FUNCTION_BLOCK FT_PT1 (* Low Pass Filter (PT1) *)
  (* Standard: 61499-1; Description: FT_PT1 is an low pass filter with a programmable time T and faktor K. *)
  (* Version 1.3, 2026-09-26, Franz Höpfinger, Bugfix (Review-Bot auf training1 PR #269, verifiziert): die neue TM.E1->RST-Verdrahtung (FT_PT1_AR v1.0) feuert RST bereits beim Start-Kaskaden-INIT (z.B. ueber initval_ATM/LatchFilterTime.INIT -> OUT.E1 -> TM.E1, siehe logiBUS_PI_Raw_Publish_OPC.SUB), also BEVOR je ein echtes REQ mit frisch abgetastetem 'in' lief. RST setzte bisher init:=TRUE UND out:=K*in mit dem zu diesem Zeitpunkt noch nie gesetzten 'in' (0.0) - das erste echte REQ sah dann init bereits TRUE und ramp'te per Euler-Schritt langsam von 0 auf den echten Wert hoch, statt sofort zu springen. RST setzt jetzt NUR NOCH init:=FALSE (kein 'in'-With-Var, kann also gar nicht sinnvoll seeden) - das naechste REQ (mit garantiert frischem 'in') macht das Seeding selbst inline (vorher this.RST(), jetzt direkt out:=K*in), genau wie beim allerersten Programmstart. *)
  (* Version 1.2, 2026-09-25, Franz Höpfinger, Bugfix (Franz live am Geraet: 'ich hatte von 2s auf 0.1s geaendert, und schwupps spinnt er' - Zapfwelle-Filterzeit auf STG4 manuell auf 100ms gesenkt): die explizite Euler-Diskretisierung wird numerisch instabil, sobald TM kleiner als das tatsaechliche REQ-Aufrufintervall (delta_t) ist - Faktor delta_t/TM > 1 laesst den Fehler pro Zyklus exponentiell wachsen statt sich dem Zielwert anzunaehern, bis out ueberlaeuft (Inf) und danach dauerhaft NaN bleibt (Inf-Inf), da kein automatisches Re-Init/RST mehr verdrahtet war. TM wird in der REQ-Berechnung jetzt adaptiv auf mindestens delta_t hochgeklemmt (Franz' Vorschlag, F1/F2-Notation) - Faktor bleibt so immer <= 1, unabhaengig von der tatsaechlichen Aufrufrate, kein fixer Magic-Number-Mindestwert noetig. *)
  (* Version 1.1, 2026-09-17, Franz Höpfinger, Bugfix (Review-Bot auf training1 PR #252, verifiziert): RST setzte init/out zurueck, aber nicht tx/last/delta_t - ein externer RST-Aufruf (jetzt ueber FT_PT1_AR.RST erreichbar) liess die naechste REQ-Ausfuehrung mit einem stehengebliebenen last einen riesigen delta_t berechnen und dadurch einen falschen Ausreisser-Schritt. RST liest jetzt T_PLC_US() neu und setzt last/delta_t entsprechend zurueck. *)
  (* Version 1.0, 2025-12-21, Franz Höpfinger, initial API and implementation and/or initial documentation *)
  PACKAGE OSCAT::Basic::POUs::Engineering::Control;
  IMPORT OSCAT::Basic::POUs::Engineering::measurements::T_PLC_US;
  IMPORT OSCAT::Basic::POUs::conversion::TIME_TO_REAL;
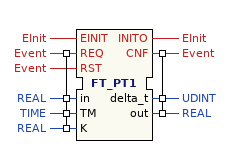
  EVENT_INPUT
    EINIT : EInit; (* Init Request *)
    REQ WITH in, TM, K; (* Normal Execution Request *)
    RST; (* Reset Filter *)
  END_EVENT
  EVENT_OUTPUT
    INITO : EInit; (* Init Confirmation *)
    CNF WITH delta_t, out; (* Execution Confirmation *)
  END_EVENT
  VAR_INPUT
    in : REAL; (* Input Signal *)
    TM : TIME; (* Filter Time Constant *)
    K : REAL := 1.0; (* Gain Factor *)
  END_VAR
  VAR_OUTPUT
    delta_t : UDINT; (* Delta T since last call. *)
    out : REAL; (* Output Signal *)
  END_VAR
  VAR
    last : UDINT; (* Last execution time *)
    tx : UDINT; (* Current execution time *)
    init : BOOL := FALSE; (* Initialization flag *)
    F1 : REAL;
    F2 : REAL;
  END_VAR
  EC_STATES
    EINIT : EINIT -> INITO; (* Initialization *)
    REQ : REQ -> CNF; (* Normal Operation *)
    RST : RST -> CNF;
  END_STATES
  ALGORITHM EINIT IN ST:
(* Reset logic *)
init := FALSE;
out := 0.0;
last := UDINT#0;
  END_ALGORITHM
  ALGORITHM RST IN ST:
(* Nur den Zustand invalidieren - das naechste REQ seedet mit frisch
   abgetastetem 'in' (With-Var, synchron zum REQ-Event). RST selbst hat
   kein 'in'-With-Var und wuerde sonst mit einem veralteten oder (beim
   allerersten Aufruf, z.B. durch TM.E1 vor der ersten echten Messung)
   noch nie gesetzten Wert (0.0) faelschlich seeden. *)
init := FALSE;
  END_ALGORITHM
  ALGORITHM REQ IN ST:
(* Read system time *)
tx := T_PLC_US();

(* Startup initialization or T=0 *)
IF NOT init OR TM = T#0s THEN
	init := TRUE;
	out := K * in;
	delta_t := UDINT#0;
ELSE
	(* Calculate time delta since last call *)
	delta_t := (tx - last);

		(* PT1 Formula: out = out + (target - out) * (dt / T) *)
	IF TIME_TO_REAL(TM) > 0.0 THEN
		F1 := UDINT_TO_REAL(delta_t) * 1.0E-3; (* delta_t in ms *)
		F2 := TIME_TO_REAL(TM); (* TM in ms *)
		IF F2 < F1 THEN
			F2 := F1;
		END_IF;
		out := out + (in * K - out) * F1 / F2;
	END_IF;

		(* Avoid denormalized numbers / underrun *)
	IF ABS(out) < 1.0E-20 THEN
		out := 0.0;
	END_IF;
END_IF;

(* Save time for next cycle *)
last := tx;
  END_ALGORITHM
END_FUNCTION_BLOCK
